// TIA Portal project "Course Work Conveyor" (V15)

(* hardware
DEVICE "S7-1200 station_1"  S7-1200 Station
   slot 0: "Rack_0"  S7-1200 Rack  Rack  V1.0
   slot 1: "PLC_1"  CPU 1214C DC/DC/DC  6ES7 214-1AG40-0XB0  V4.0
   slot 3: "AQ 1x12BIT_1"  AQ1 signal board  6ES7 232-4HA30-0XB0  V1.0
DEVICE "HMI_1"  KTP700 Basic PN
   slot 0: "HMI_1"  KTP700 Basic PN  6AV2 123-2GB03-0AX0  15.0.0.0
   slot 1: "HMI_RT_1"  KTP700 Basic PN  6AV2 123-2GB03-0AX0  15.0.0.0
   slot 5: "HMI_1.IE_CP_1"  PROFINET Interface  15.0.0.0
      slot 1: "PROFINET Interface_1"  PROFINET Interface
         slot 1: "Port_1"  Port
*)

// ===== PLC "PLC_1"  CPU 1214C DC/DC/DC =====

VAR_GLOBAL   // PLC tag table "Input/Output/Bit Tag Table"
   "EMS" AT %I0.0 : Bool;   // Emergency Stop Button NC (Input)
   "S1_Optical" AT %I0.1 : Bool;   // Optical Start Conveyor Sensor - NO (Input)
   "S2_Optical" AT %I0.2 : Bool;   // Optical Check Size Sensor NO (Input)
   "S3_Heat_or_Reject" AT %I0.3 : Bool;   // Optical Heat or Reject position Sensor NO (Input)
   "Temperature_Read_in" AT %IW64 : Int;   // Analogue Temperature (Input)
   "Reject" AT %Q0.0 : Bool;   // Rejection Solenoid (Output)
   "Conveyor" AT %Q0.1 : Bool;   // Conveyor Run (Output)
   "Furnace" AT %Q0.2 : Bool;   // Furnace Heater (Output)
   "System_Enable" AT %M0.0 : Bool;   // System Enable (Bit)
   "Detected_Large" AT %M0.1 : Bool;   // Large piece (Detected) (Bit)
   "Detected_Small" AT %M0.2 : Bool;   // Small piece (Detected) (Bit)
   "Reject_for_Large" AT %M0.5 : Bool;   // Large Rejection (Selected) (Bit)
   "Reject_for_Small" AT %M0.4 : Bool;   // Small Rejection (Selected) (Bit)
   "Furnace_Enable" AT %M0.6 : Bool;   // Furnace conditions met (Bit)
   "Piece_Size_Reset" AT %M0.7 : Bool;   // Reset the basket size (Bit)
   "PV_Memory" AT %MD1 : Real;   // Present Value reading word (Word byte)
   "Temp_in_Range" AT %M11.0 : Bool;   // Temperature in Range Confirmation (Bit)
   "Auto_Stop_Reset" AT %M11.2 : Bool;   // Automatic Stop and Reset for errors (Bit)
   "Temp_High_Alarm" AT %M11.3 : Bool;   // Furnace Alarm Temperature too High (Bit)
   "Temp_Low_Alarm" AT %M11.4 : Bool;   // Furnace Alarm Temperature too Low (Bit)
   "Temp_High_Set_Point" AT %MD12 : Real;   // High Temperature Setpoint (Bit)
   "Temp_Low_Set_Point" AT %MD16 : Real;   // Low Temperature Setpoint (Bit)
   "Temp_Limit_High_Range" AT %MD20 : Real;   // Temperature range confirmation High (Bit)
   "Temp_Limit_Low_Range" AT %MD24 : Real;   // Temperature range confirmation Low (Bit)
   "Furnace_Cycle_end" AT %M28.0 : Bool;   // End of Furnace cycle (Bit)
   "Piece_selected" AT %M28.3 : Bool;   // Confirms a piece size has been selected. (Bit)
   "Piece_Detected" AT %M28.4 : Bool;   // Confirms a piece has been detected.(Bit)
   "Counter_Reset_Large" AT %M28.5 : Bool;   // Large Piece Counter Reset (Bit)
   "Counter_Reset_Small" AT %M28.6 : Bool;   // Small Piece Counter Reset (Bit)
   "Counter_Reset_Errors" AT %M28.7 : Bool;   // Error Counter Reset (Bit)
   "Counter_Reset_Rejects" AT %M29.0 : Bool;   // Piece Reject Counter Reset (Bit)
END_VAR

VAR_GLOBAL   // PLC tag table "HMI Control Tag Table"
   "PB_Furnace_Activation_HMI" AT %M10.7 : Bool;   // Push Button: to Activate PID control of Furnace NO (Input)
   "PB_Small_HMI" AT %M10.0 : Bool;   // Push Button: Small Size reject NO (Input)
   "PB_Large_HMI" AT %M10.2 : Bool;   // Push Button: Large Size reject NO (Input)
   "PB_Manual_HMI" AT %M10.3 : Bool;   // Push Button: Mode Manual Selected NO (Input)
   "PB_Automatic_HMI" AT %M10.4 : Bool;   // Push Button: Mode Automatic Selected NO (Input)
   "PB_Reject_All_HMI" AT %M10.5 : Bool;   // Push Button: Reject All Size of Pieces NO (Input)
   "PB_Stop_Reset_HMI" AT %M10.6 : Bool;   // Push Button: Stop/Reset process cycle NO (Input)
   "PB_Furnace_Deactivation_HMI" AT %M11.1 : Bool;   // Push Button: to deactivate PID control of Furnace NO (Input)
   "PB_Reset_Counter_Large_HMI" AT %M11.5 : Bool;   // Push Button: to reset the large piece counter NO (Input)
   "PB_Reset_Counter_Small_HMI" AT %M11.6 : Bool;   // Push Button: to reset the small piece counter NO (Input)
   "PB_Reset_Counter_Errors_HMI" AT %M11.7 : Bool;   // Push Button: to reset the error counter NO (Input)
   "PB_Reset_Counter_Rejects_HMI" AT %M28.1 : Bool;   // Push Button: to reset the rejects counter NO (Input)
   "PB_Reset_Counter_All_HMI" AT %M28.2 : Bool;   // Push Button: to reset all the counters NO (Input)
   "Piece_inserted_Error_Light_HMI" AT %M29.1 : Bool;   // Error Light on HMI for Piece inserted before end the of cycle (Output)
END_VAR

DATA_BLOCK "Temp_Analog_In_DB"   // DB2
{ S7_Optimized_Access := 'TRUE' }
VERSION : 0.1
// stored: InstanceOfName Temp_Analog_In
"Temp_Analog_In"
BEGIN
END_DATA_BLOCK

// folder: System blocks/Program resources

DATA_BLOCK "Piece_Size_Reset_Delay_Timer_0_DB_2"   // DB3
{ S7_Optimized_Access := 'TRUE' }
AUTHOR : Simatic
FAMILY : IEC
NAME : IEC_TMR
VERSION : 1.0
// stored: InstanceOfName IEC_TIMER
"IEC_TIMER"
BEGIN
END_DATA_BLOCK

DATA_BLOCK "Small_Piece_Counter_0_DB"   // DB7
{ S7_Optimized_Access := 'TRUE' }
AUTHOR : Simatic
FAMILY : IEC
NAME : CNTR
VERSION : 1.0
// stored: InstanceOfName IEC_COUNTER
"IEC_COUNTER"
BEGIN
END_DATA_BLOCK

DATA_BLOCK "Large_Piece_Counter_0_DB"   // DB8
{ S7_Optimized_Access := 'TRUE' }
AUTHOR : Simatic
FAMILY : IEC
NAME : CNTR
VERSION : 1.0
// stored: InstanceOfName IEC_COUNTER
"IEC_COUNTER"
BEGIN
END_DATA_BLOCK

DATA_BLOCK "Furnace_Timer_0_DB_2"   // DB9
{ S7_Optimized_Access := 'TRUE' }
AUTHOR : Simatic
FAMILY : IEC
NAME : IEC_TMR
VERSION : 1.0
// stored: InstanceOfName IEC_TIMER
"IEC_TIMER"
BEGIN
END_DATA_BLOCK

DATA_BLOCK "Total_Error_Counter_0_DB"   // DB10
{ S7_Optimized_Access := 'TRUE' }
AUTHOR : Simatic
FAMILY : IEC
NAME : CNTR
VERSION : 1.0
// stored: InstanceOfName IEC_COUNTER
"IEC_COUNTER"
BEGIN
END_DATA_BLOCK

DATA_BLOCK "Total_Piece_Reject_Counter_0_DB"   // DB11
{ S7_Optimized_Access := 'TRUE' }
AUTHOR : Simatic
FAMILY : IEC
NAME : CNTR
VERSION : 1.0
// stored: InstanceOfName IEC_COUNTER
"IEC_COUNTER"
BEGIN
END_DATA_BLOCK

DATA_BLOCK "Reject_on_Error_Delay_Timer_0_DB_3"   // DB12
{ S7_Optimized_Access := 'TRUE' }
AUTHOR : Simatic
FAMILY : IEC
NAME : IEC_TMR
VERSION : 1.0
// stored: InstanceOfName IEC_TIMER
"IEC_TIMER"
BEGIN
END_DATA_BLOCK

// folder: (top level)

FUNCTION_BLOCK "Temp_Analog_In"   // FB1, LAD
{ S7_Optimized_Access := 'TRUE' }
VERSION : 0.1
// Function Block: Temperature (Analogue Signal In). 
// The Temperature signal is read, normalised and then put to scale.
   VAR_INPUT
      ChannelAddress : Int;
      HR : Real;
      LR : Real;
   END_VAR
   VAR_IN_OUT
      PV : Real;   // Input reading
   END_VAR
   VAR_TEMP
      Normalised : Real;   // Normalise Temperature Value
   END_VAR
BEGIN

REGION Network 1: Value Normalising.
   // Normalising reading values (Scale 0 to 27648).
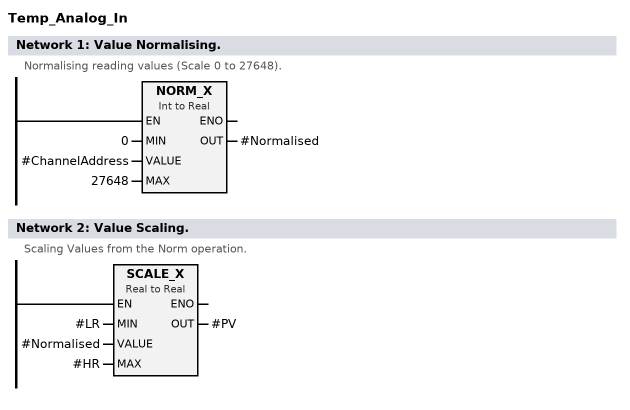
   RUNG wire#powerrail
      { S7_Templates := "[SrcType := Int, DestType := Real]" } Normalize(min := 0, value := #ChannelAddress, max := 27648, out => #Normalised)
   END_RUNG
   // the same network as SCL:
   #Normalised := NORM_X(MIN := 0, VALUE := #ChannelAddress, MAX := 27648);
END_REGION

REGION Network 2: Value Scaling.
   // Scaling Values from the Norm operation.
   RUNG wire#powerrail
      { S7_Templates := "[SrcType := Real, DestType := Real]" } Scale(min := #LR, value := #Normalised, max := #HR, out => #PV)
   END_RUNG
   // the same network as SCL:
   #PV := SCALE_X(MIN := #LR, VALUE := #Normalised, MAX := #HR);
END_REGION
END_FUNCTION_BLOCK

FUNCTION "Conveyor Belt" : Void   // FC1, LAD
{ S7_Optimized_Access := 'TRUE' }
VERSION : 0.1
// Conveyor Related Operations:
// Conveyor Run.
// Piece Size Detection.
// Piece size Confirmation.
// Rejection Solenoid.
// Enable Furnace Operation.
// Furnace in Operation.
// Basket Size Reset.
BEGIN

REGION Network 1: Conveyor Run
   // Once size is selected AND System is Enabled (Automatic mode) OR Manual == Conveyor ON
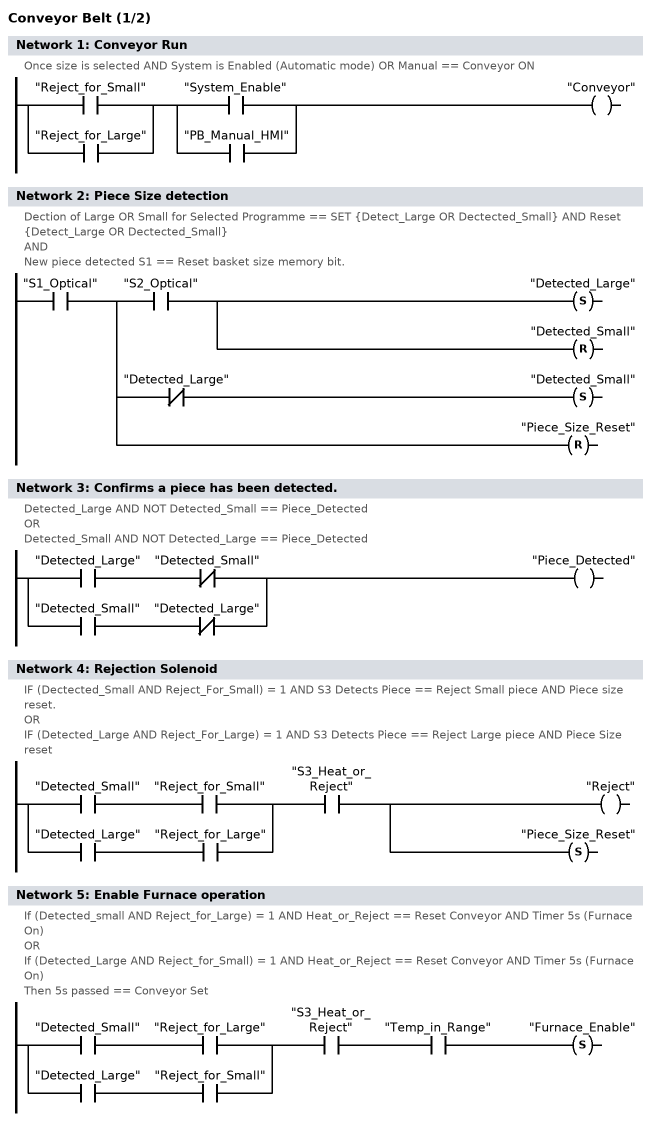
   RUNG wire#powerrail
      Contact( "Reject_for_Small" )
      wire#w1
      Contact( "System_Enable" )
      wire#w2
      Coil( "Conveyor" )
   END_RUNG
   RUNG wire#powerrail
      Contact( "Reject_for_Large" )
   END_RUNG wire#w1
   RUNG wire#w1
      Contact( "PB_Manual_HMI" )
   END_RUNG wire#w2
   // the same network as SCL:
   "Conveyor" := ("Reject_for_Small" OR "Reject_for_Large") AND ("System_Enable" OR "PB_Manual_HMI");
END_REGION

REGION Network 2: Piece Size detection
   // Dection of Large OR Small for Selected Programme == SET {Detect_Large OR Dectected_Small} AND Reset {Detect_Large OR Dectected_Small}
   // AND
   // New piece detected S1 == Reset basket size memory bit.
   RUNG wire#powerrail
      Contact( "S1_Optical" )
      wire#w1
      Contact( "S2_Optical" )
      wire#w2
      S_Coil( "Detected_Large" )
   END_RUNG
   RUNG wire#w2
      R_Coil( "Detected_Small" )
   END_RUNG
   RUNG wire#w1
      I_Contact( "Detected_Large" )
      S_Coil( "Detected_Small" )
   END_RUNG
   RUNG wire#w1
      R_Coil( "Piece_Size_Reset" )
   END_RUNG
   // the same network as SCL:
   IF "S1_Optical" AND "S2_Optical" THEN
       "Detected_Large" := TRUE;
       "Detected_Small" := FALSE;
   END_IF;
   IF "S1_Optical" AND NOT "Detected_Large" THEN "Detected_Small" := TRUE; END_IF;
   IF "S1_Optical" THEN "Piece_Size_Reset" := FALSE; END_IF;
END_REGION

REGION Network 3: Confirms a piece has been detected.
   // Detected_Large AND NOT Detected_Small == Piece_Detected
   // OR
   // Detected_Small AND NOT Detected_Large == Piece_Detected
   RUNG wire#powerrail
      Contact( "Detected_Large" )
      I_Contact( "Detected_Small" )
      wire#w1
      Coil( "Piece_Detected" )
   END_RUNG
   RUNG wire#powerrail
      Contact( "Detected_Small" )
      I_Contact( "Detected_Large" )
   END_RUNG wire#w1
   // the same network as SCL:
   "Piece_Detected" := ("Detected_Large" AND NOT "Detected_Small") OR ("Detected_Small" AND NOT "Detected_Large");
END_REGION

REGION Network 4: Rejection Solenoid
   // IF (Dectected_Small AND Reject_For_Small) = 1 AND S3 Detects Piece == Reject Small piece AND Piece size reset.
   // OR
   // IF (Detected_Large AND Reject_For_Large) = 1 AND S3 Detects Piece == Reject Large piece AND Piece Size reset
   RUNG wire#powerrail
      Contact( "Detected_Small" )
      Contact( "Reject_for_Small" )
      wire#w1
      Contact( "S3_Heat_or_Reject" )
      wire#w2
      Coil( "Reject" )
   END_RUNG
   RUNG wire#powerrail
      Contact( "Detected_Large" )
      Contact( "Reject_for_Large" )
   END_RUNG wire#w1
   RUNG wire#w2
      S_Coil( "Piece_Size_Reset" )
   END_RUNG
   // the same network as SCL:
   "Reject" := (("Detected_Small" AND "Reject_for_Small") OR ("Detected_Large" AND "Reject_for_Large")) AND "S3_Heat_or_Reject";
   IF "Reject" THEN "Piece_Size_Reset" := TRUE; END_IF;
END_REGION

REGION Network 5: Enable Furnace operation
   // If (Detected_small AND Reject_for_Large) = 1 AND Heat_or_Reject == Reset Conveyor AND Timer 5s (Furnace On)
   // OR
   // If (Detected_Large AND Reject_for_Small) = 1 AND Heat_or_Reject == Reset Conveyor AND Timer 5s (Furnace On)
   // Then 5s passed == Conveyor Set
   RUNG wire#powerrail
      Contact( "Detected_Small" )
      Contact( "Reject_for_Large" )
      wire#w1
      Contact( "S3_Heat_or_Reject" )
      Contact( "Temp_in_Range" )
      S_Coil( "Furnace_Enable" )
   END_RUNG
   RUNG wire#powerrail
      Contact( "Detected_Large" )
      Contact( "Reject_for_Small" )
   END_RUNG wire#w1
   // the same network as SCL:
   IF (("Detected_Small" AND "Reject_for_Large") OR ("Detected_Large" AND "Reject_for_Small")) AND "S3_Heat_or_Reject" AND "Temp_in_Range" THEN
       "Furnace_Enable" := TRUE;
   END_IF;
END_REGION

REGION Network 6: Furnace in Operation
   // IF Furnace enabled == stop Conveyor 
   // THEN  Temp_in_Range == start 5s Timer
   // AND THEN at 5s == reset Conveyor AND Reset_Piece_Size AND SET  Furnace_Cycle_end
   // Note: Timer delay on piece size reset to allow and of cycle tasks before new cycle.
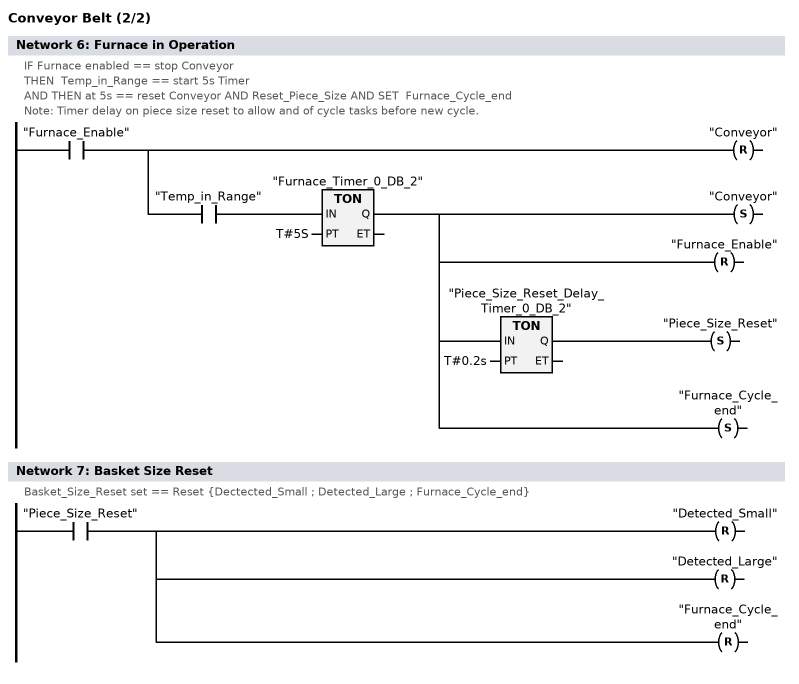
   IF "Furnace_Enable" THEN "Conveyor" := FALSE; END_IF;
   "Furnace_Timer_0_DB_2".TON(IN := "Furnace_Enable" AND "Temp_in_Range", PT := T#5S);
   IF "Furnace_Timer_0_DB_2".Q THEN
       "Conveyor" := TRUE;
       "Furnace_Enable" := FALSE;
   END_IF;
   "Piece_Size_Reset_Delay_Timer_0_DB_2".TON(IN := "Furnace_Timer_0_DB_2".Q, PT := T#0.2s);
   IF "Piece_Size_Reset_Delay_Timer_0_DB_2".Q THEN "Piece_Size_Reset" := TRUE; END_IF;
   IF "Furnace_Timer_0_DB_2".Q THEN "Furnace_Cycle_end" := TRUE; END_IF;
END_REGION

REGION Network 7: Basket Size Reset
   // Basket_Size_Reset set == Reset {Dectected_Small ; Detected_Large ; Furnace_Cycle_end}
   RUNG wire#powerrail
      Contact( "Piece_Size_Reset" )
      wire#w1
      R_Coil( "Detected_Small" )
   END_RUNG
   RUNG wire#w1
      R_Coil( "Detected_Large" )
   END_RUNG
   RUNG wire#w1
      R_Coil( "Furnace_Cycle_end" )
   END_RUNG
   // the same network as SCL:
   IF "Piece_Size_Reset" THEN
       "Detected_Small" := FALSE;
       "Detected_Large" := FALSE;
       "Furnace_Cycle_end" := FALSE;
   END_IF;
END_REGION
END_FUNCTION

FUNCTION "Temperature Function" : Void   // FC2, LAD
{ S7_Optimized_Access := 'TRUE' }
VERSION : 0.1
BEGIN

REGION Network 1: PID Control of the Furnace Activation/Deactivation
   // IF Button "Funace Activation" pressed == PID Control ON
   // OR
   // IF Button "Stop Furnace" pressed == PID Control OFF
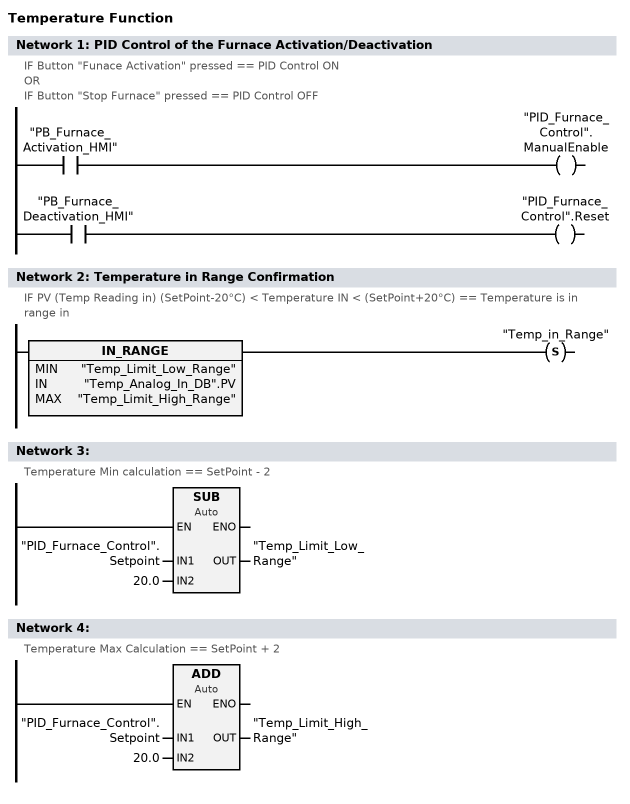
   RUNG wire#powerrail
      Contact( "PB_Furnace_Activation_HMI" )
      Coil( "PID_Furnace_Control".ManualEnable )
   END_RUNG
   RUNG wire#powerrail
      Contact( "PB_Furnace_Deactivation_HMI" )
      Coil( "PID_Furnace_Control".Reset )
   END_RUNG
   // the same network as SCL:
   "PID_Furnace_Control".ManualEnable := "PB_Furnace_Activation_HMI";
   "PID_Furnace_Control".Reset := "PB_Furnace_Deactivation_HMI";
END_REGION

REGION Network 2: Temperature in Range Confirmation
   // IF PV (Temp Reading in) (SetPoint-20°C) < Temperature IN < (SetPoint+20°C) == Temperature is in range in
   RUNG wire#powerrail
      { S7_Templates := "SrcType := Real" } InRange(min := "Temp_Limit_Low_Range", in := "Temp_Analog_In_DB".PV, max := "Temp_Limit_High_Range")
      S_Coil( "Temp_in_Range" )
   END_RUNG
   // the same network as SCL:
   IF ("Temp_Limit_Low_Range" <= "Temp_Analog_In_DB".PV) AND ("Temp_Analog_In_DB".PV <= "Temp_Limit_High_Range") THEN
       "Temp_in_Range" := TRUE;
   END_IF;
END_REGION

REGION Network 3
   // Temperature Min calculation == SetPoint - 2
   RUNG wire#powerrail
      Sub(in1 := "PID_Furnace_Control".Setpoint, in2 := 20.0, out => "Temp_Limit_Low_Range")
   END_RUNG
   // the same network as SCL:
   "Temp_Limit_Low_Range" := "PID_Furnace_Control".Setpoint - 20.0;
END_REGION

REGION Network 4
   // Temperature Max Calculation == SetPoint + 2
   RUNG wire#powerrail
      Add(in1 := "PID_Furnace_Control".Setpoint, in2 := 20.0, out => "Temp_Limit_High_Range")
   END_RUNG
   // the same network as SCL:
   "Temp_Limit_High_Range" := "PID_Furnace_Control".Setpoint + 20.0;
END_REGION
END_FUNCTION

FUNCTION "Error_Handling" : Void   // FC3, LAD
{ S7_Optimized_Access := 'TRUE' }
VERSION : 0.1
// Error Handling Function:
// Piece inserted before end of previous cycle
// Temperature is Too HIGH or too LOW.
   VAR_TEMP   // added for the SCL form of the ladder/FBD networks
      _w1 : Bool;
   END_VAR
BEGIN

REGION Network 1: Rejection Solenoid
   // Piece inserted before end of previous cycle:
   // Piece detected at Heating/Rejection point AND (S1 OR S2) triggered == Reject Part AND Stop/Reset Cycle AND Sets the Error Light ON on the HMI.
   // Note: The Timer delays the reject to leave time for Auto_Stop_Reset and the Error Light to set ON.
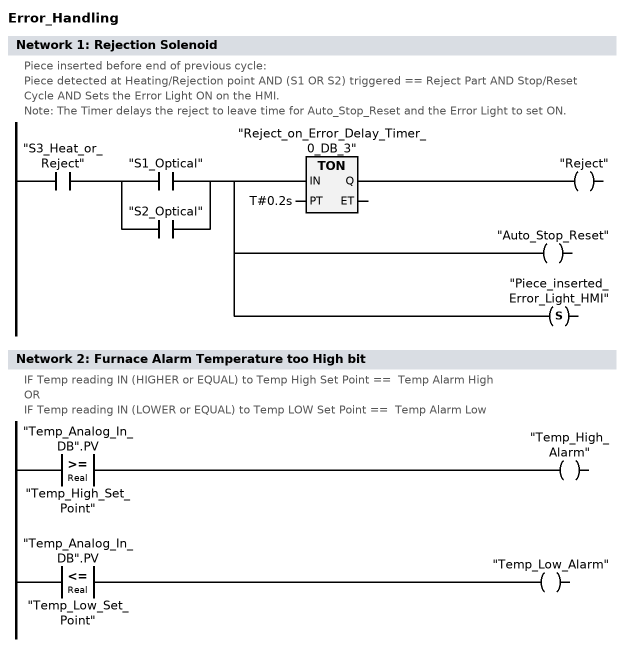
   #_w1 := "S3_Heat_or_Reject" AND ("S1_Optical" OR "S2_Optical");
   "Reject_on_Error_Delay_Timer_0_DB_3".TON(IN := #_w1, PT := T#0.2s);
   "Reject" := "Reject_on_Error_Delay_Timer_0_DB_3".Q;
   "Auto_Stop_Reset" := #_w1;
   IF #_w1 THEN "Piece_inserted_Error_Light_HMI" := TRUE; END_IF;
END_REGION

REGION Network 2: Furnace Alarm Temperature too High bit
   // IF Temp reading IN (HIGHER or EQUAL) to Temp High Set Point ==  Temp Alarm High
   // OR
   // IF Temp reading IN (LOWER or EQUAL) to Temp LOW Set Point ==  Temp Alarm Low
   RUNG wire#powerrail
      { S7_Templates := "SrcType := Real" } GE_Contact(in1 := "Temp_Analog_In_DB".PV, in2 := "Temp_High_Set_Point")
      Coil( "Temp_High_Alarm" )
   END_RUNG
   RUNG wire#powerrail
      { S7_Templates := "SrcType := Real" } LE_Contact(in1 := "Temp_Analog_In_DB".PV, in2 := "Temp_Low_Set_Point")
      Coil( "Temp_Low_Alarm" )
   END_RUNG
   // the same network as SCL:
   "Temp_High_Alarm" := "Temp_Analog_In_DB".PV >= "Temp_High_Set_Point";
   "Temp_Low_Alarm" := "Temp_Analog_In_DB".PV <= "Temp_Low_Set_Point";
END_REGION
END_FUNCTION

FUNCTION "Counters" : Void   // FC4, LAD
{ S7_Optimized_Access := 'TRUE' }
VERSION : 0.1
// Counters in the process for each manufactured parts and for the number of errors.
BEGIN

REGION Network 1: Large part manufactured counter.
   // IF Detected_Large AND Reject_for_small AND Furnace_Cycle_end == Counter +1
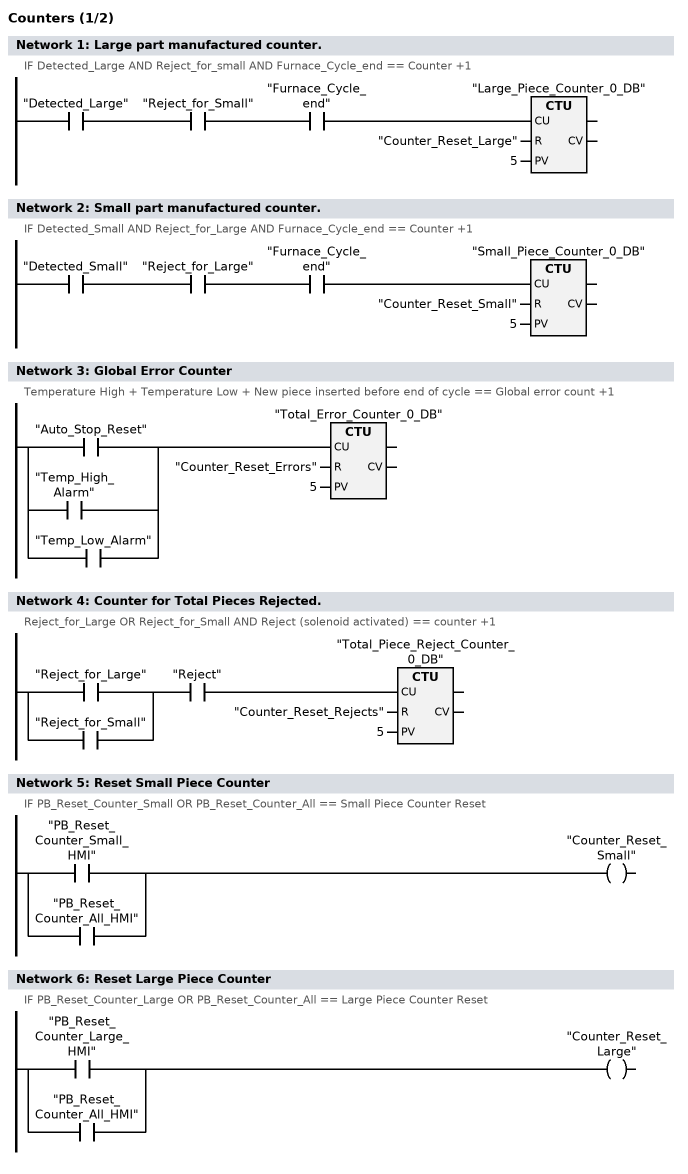
   "Large_Piece_Counter_0_DB".CTU(CU := "Detected_Large" AND "Reject_for_Small" AND "Furnace_Cycle_end",
                           R := "Counter_Reset_Large",
                           PV := 5);
END_REGION

REGION Network 2: Small part manufactured counter.
   // IF Detected_Small AND Reject_for_Large AND Furnace_Cycle_end == Counter +1
   "Small_Piece_Counter_0_DB".CTU(CU := "Detected_Small" AND "Reject_for_Large" AND "Furnace_Cycle_end",
                           R := "Counter_Reset_Small",
                           PV := 5);
END_REGION

REGION Network 3: Global Error Counter
   // Temperature High + Temperature Low + New piece inserted before end of cycle == Global error count +1
   "Total_Error_Counter_0_DB".CTU(CU := "Auto_Stop_Reset" OR "Temp_High_Alarm" OR "Temp_Low_Alarm",
                           R := "Counter_Reset_Errors",
                           PV := 5);
END_REGION

REGION Network 4: Counter for Total Pieces Rejected.
   // Reject_for_Large OR Reject_for_Small AND Reject (solenoid activated) == counter +1
   "Total_Piece_Reject_Counter_0_DB".CTU(CU := ("Reject_for_Large" OR "Reject_for_Small") AND "Reject",
                           R := "Counter_Reset_Rejects",
                           PV := 5);
END_REGION

REGION Network 5: Reset Small Piece Counter
   // IF PB_Reset_Counter_Small OR PB_Reset_Counter_All == Small Piece Counter Reset
   RUNG wire#powerrail
      Contact( "PB_Reset_Counter_Small_HMI" )
      wire#w1
      Coil( "Counter_Reset_Small" )
   END_RUNG
   RUNG wire#powerrail
      Contact( "PB_Reset_Counter_All_HMI" )
   END_RUNG wire#w1
   // the same network as SCL:
   "Counter_Reset_Small" := "PB_Reset_Counter_Small_HMI" OR "PB_Reset_Counter_All_HMI";
END_REGION

REGION Network 6: Reset Large Piece Counter
   // IF PB_Reset_Counter_Large OR PB_Reset_Counter_All == Large Piece Counter Reset
   RUNG wire#powerrail
      Contact( "PB_Reset_Counter_Large_HMI" )
      wire#w1
      Coil( "Counter_Reset_Large" )
   END_RUNG
   RUNG wire#powerrail
      Contact( "PB_Reset_Counter_All_HMI" )
   END_RUNG wire#w1
   // the same network as SCL:
   "Counter_Reset_Large" := "PB_Reset_Counter_Large_HMI" OR "PB_Reset_Counter_All_HMI";
END_REGION

REGION Network 7: Reset Rejected Piece Counter
   // IF PB_Reset_Counter_Reject OR PB_Reset_Counter_All == Total Piece Rejects Counter Reset
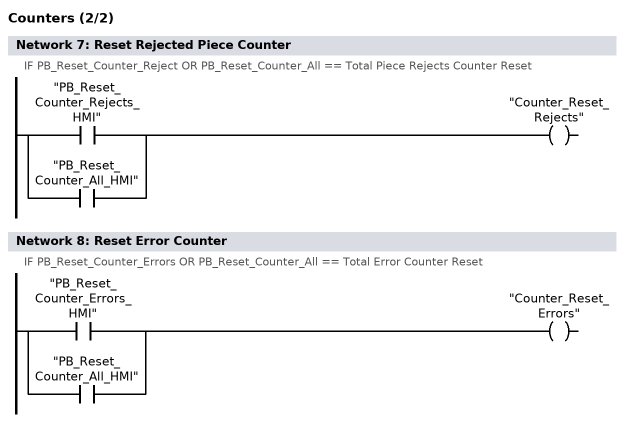
   RUNG wire#powerrail
      Contact( "PB_Reset_Counter_Rejects_HMI" )
      wire#w1
      Coil( "Counter_Reset_Rejects" )
   END_RUNG
   RUNG wire#powerrail
      Contact( "PB_Reset_Counter_All_HMI" )
   END_RUNG wire#w1
   // the same network as SCL:
   "Counter_Reset_Rejects" := "PB_Reset_Counter_Rejects_HMI" OR "PB_Reset_Counter_All_HMI";
END_REGION

REGION Network 8: Reset Error Counter
   // IF PB_Reset_Counter_Errors OR PB_Reset_Counter_All == Total Error Counter Reset
   RUNG wire#powerrail
      Contact( "PB_Reset_Counter_Errors_HMI" )
      wire#w1
      Coil( "Counter_Reset_Errors" )
   END_RUNG
   RUNG wire#powerrail
      Contact( "PB_Reset_Counter_All_HMI" )
   END_RUNG wire#w1
   // the same network as SCL:
   "Counter_Reset_Errors" := "PB_Reset_Counter_Errors_HMI" OR "PB_Reset_Counter_All_HMI";
END_REGION
END_FUNCTION

FUNCTION "System_Controls" : Void   // FC5, LAD
TITLE = Systems_Controls
{ S7_Optimized_Access := 'TRUE' }
VERSION : 0.1
// Interface controls to enable the automatic mode.
// Stop/Reset on HMI and auto Reset operations.
// Piece size selection and confirmation operation.
BEGIN

REGION Network 1: Automatic Mode System Enable
   // Automatic Mode && Part Detected AND Temp in Range AND NOT Manual mode  == System enabled AND Error_Light for piece inserted reset.
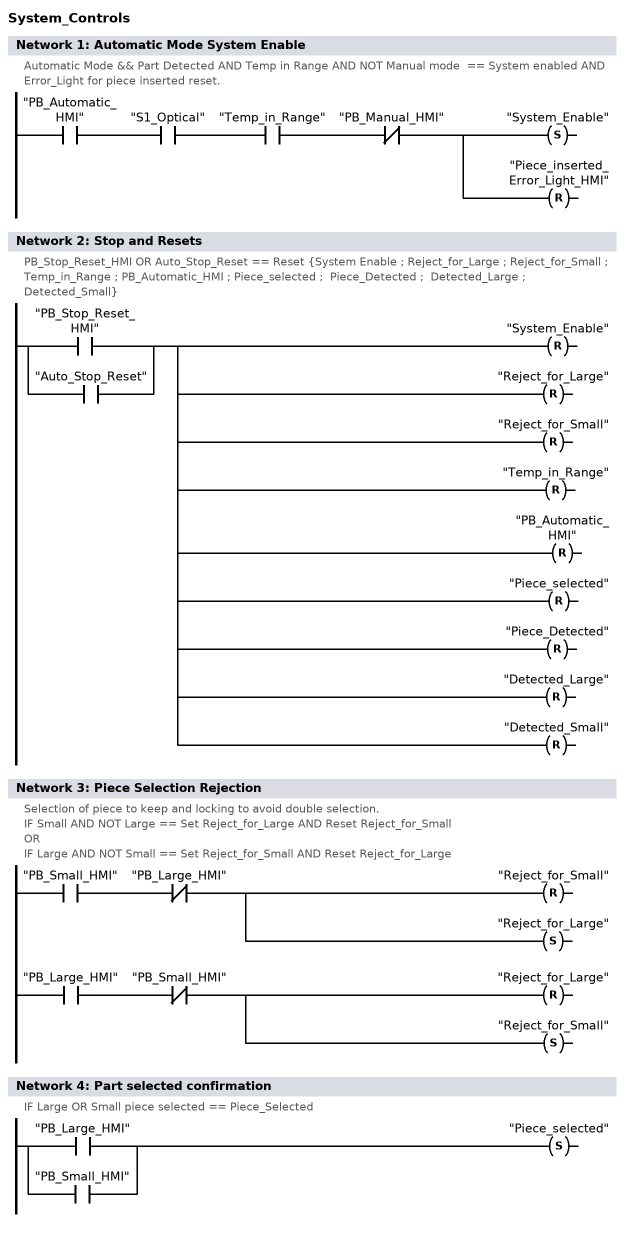
   RUNG wire#powerrail
      Contact( "PB_Automatic_HMI" )
      Contact( "S1_Optical" )
      Contact( "Temp_in_Range" )
      I_Contact( "PB_Manual_HMI" )
      wire#w1
      S_Coil( "System_Enable" )
   END_RUNG
   RUNG wire#w1
      R_Coil( "Piece_inserted_Error_Light_HMI" )
   END_RUNG
   // the same network as SCL:
   IF "PB_Automatic_HMI" AND "S1_Optical" AND "Temp_in_Range" AND NOT "PB_Manual_HMI" THEN
       "System_Enable" := TRUE;
       "Piece_inserted_Error_Light_HMI" := FALSE;
   END_IF;
END_REGION

REGION Network 2: Stop and Resets
   // PB_Stop_Reset_HMI OR Auto_Stop_Reset == Reset {System Enable ; Reject_for_Large ; Reject_for_Small ; Temp_in_Range ; PB_Automatic_HMI ; Piece_selected ;  Piece_Detected ;  Detected_Large ; Detected_Small}
   RUNG wire#powerrail
      Contact( "PB_Stop_Reset_HMI" )
      wire#w1
      R_Coil( "System_Enable" )
   END_RUNG
   RUNG wire#powerrail
      Contact( "Auto_Stop_Reset" )
   END_RUNG wire#w1
   RUNG wire#w1
      R_Coil( "Reject_for_Large" )
   END_RUNG
   RUNG wire#w1
      R_Coil( "Reject_for_Small" )
   END_RUNG
   RUNG wire#w1
      R_Coil( "Temp_in_Range" )
   END_RUNG
   RUNG wire#w1
      R_Coil( "PB_Automatic_HMI" )
   END_RUNG
   RUNG wire#w1
      R_Coil( "Piece_selected" )
   END_RUNG
   RUNG wire#w1
      R_Coil( "Piece_Detected" )
   END_RUNG
   RUNG wire#w1
      R_Coil( "Detected_Large" )
   END_RUNG
   RUNG wire#w1
      R_Coil( "Detected_Small" )
   END_RUNG
   // the same network as SCL:
   IF "PB_Stop_Reset_HMI" OR "Auto_Stop_Reset" THEN
       "System_Enable" := FALSE;
       "Reject_for_Large" := FALSE;
       "Reject_for_Small" := FALSE;
       "Temp_in_Range" := FALSE;
       "PB_Automatic_HMI" := FALSE;
       "Piece_selected" := FALSE;
       "Piece_Detected" := FALSE;
       "Detected_Large" := FALSE;
       "Detected_Small" := FALSE;
   END_IF;
END_REGION

REGION Network 3: Piece Selection Rejection
   // Selection of piece to keep and locking to avoid double selection. 
   // IF Small AND NOT Large == Set Reject_for_Large AND Reset Reject_for_Small
   // OR
   // IF Large AND NOT Small == Set Reject_for_Small AND Reset Reject_for_Large
   RUNG wire#powerrail
      Contact( "PB_Small_HMI" )
      I_Contact( "PB_Large_HMI" )
      wire#w1
      R_Coil( "Reject_for_Small" )
   END_RUNG
   RUNG wire#w1
      S_Coil( "Reject_for_Large" )
   END_RUNG
   RUNG wire#powerrail
      Contact( "PB_Large_HMI" )
      I_Contact( "PB_Small_HMI" )
      wire#w2
      R_Coil( "Reject_for_Large" )
   END_RUNG
   RUNG wire#w2
      S_Coil( "Reject_for_Small" )
   END_RUNG
   // the same network as SCL:
   IF "PB_Small_HMI" AND NOT "PB_Large_HMI" THEN
       "Reject_for_Small" := FALSE;
       "Reject_for_Large" := TRUE;
   END_IF;
   IF "PB_Large_HMI" AND NOT "PB_Small_HMI" THEN
       "Reject_for_Large" := FALSE;
       "Reject_for_Small" := TRUE;
   END_IF;
END_REGION

REGION Network 4: Part selected confirmation
   // IF Large OR Small piece selected == Piece_Selected
   RUNG wire#powerrail
      Contact( "PB_Large_HMI" )
      wire#w1
      S_Coil( "Piece_selected" )
   END_RUNG
   RUNG wire#powerrail
      Contact( "PB_Small_HMI" )
   END_RUNG wire#w1
   // the same network as SCL:
   IF "PB_Large_HMI" OR "PB_Small_HMI" THEN "Piece_selected" := TRUE; END_IF;
END_REGION
END_FUNCTION

ORGANIZATION_BLOCK "Main"   // OB1, LAD, ProgramCycle
TITLE = "Main Program Sweep (Cycle)"
{ S7_Optimized_Access := 'TRUE' }
VERSION : 0.1
// Main loop of the Programme. It contains:
// The System Controls and Conveyor Belt operation
// The read in value from the analogue temperature sensor.
// The Counter function.
   VAR_INPUT
      Initial_Call : Bool;   // Initial call of this OB
      Remanence : Bool;   // =True, if remanent data are available
   END_VAR
   VAR_TEMP   // added for the SCL form of the ladder/FBD networks
      _w1 : Bool;
   END_VAR
BEGIN

REGION Network 1: Programme main functions
   // System_Controls: Link with the HMI interface.  Allows piece sizes selection and programme selection (Automatic or Manual)
   // Conveyor Belt:  Conveyor belt, piece rejection and furnace operation.
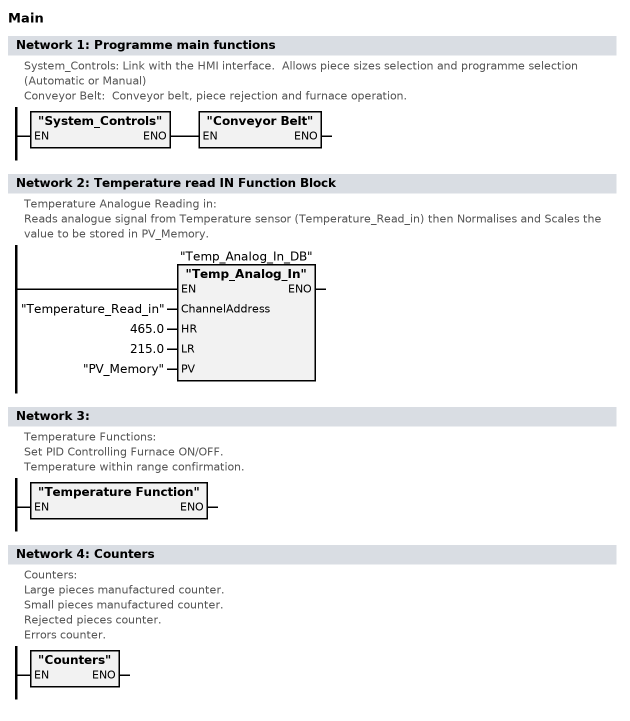
   RUNG wire#powerrail
      "System_Controls"()
      "Conveyor Belt"()
   END_RUNG
   // the same network as SCL:
   "System_Controls"(ENO => #_w1);
   IF #_w1 THEN "Conveyor Belt"(); END_IF;
END_REGION

REGION Network 2: Temperature read IN Function Block
   // Temperature Analogue Reading in:
   // Reads analogue signal from Temperature sensor (Temperature_Read_in) then Normalises and Scales the value to be stored in PV_Memory.
   RUNG wire#powerrail
      "Temp_Analog_In_DB"(ChannelAddress := "Temperature_Read_in", HR := 465.0, LR := 215.0, PV := "PV_Memory")
   END_RUNG
   // the same network as SCL:
   "Temp_Analog_In_DB"(ChannelAddress := "Temperature_Read_in", HR := 465.0, LR := 215.0, PV := "PV_Memory");   // "Temp_Analog_In"
END_REGION

REGION Network 3
   // Temperature Functions: 
   // Set PID Controlling Furnace ON/OFF.
   // Temperature within range confirmation.
   RUNG wire#powerrail
      "Temperature Function"()
   END_RUNG
   // the same network as SCL:
   "Temperature Function"();
END_REGION

REGION Network 4: Counters
   // Counters:
   // Large pieces manufactured counter.
   // Small pieces manufactured counter.
   // Rejected pieces counter.
   // Errors counter.
   RUNG wire#powerrail
      "Counters"()
   END_RUNG
   // the same network as SCL:
   "Counters"();
END_REGION
END_ORGANIZATION_BLOCK

ORGANIZATION_BLOCK "Cyclic interrupt"   // OB30, LAD, CyclicInterrupt
{ S7_Optimized_Access := 'TRUE' }
VERSION : 0.1
// OB30 allows for background tasks to run at the same time time as the main programme:
// Furnace PID Control.
// Error Handling function.
   VAR_INPUT
      Initial_Call : Bool;   // Initial call of this OB
      Event_Count : Int;   // Events discarded
   END_VAR
BEGIN

REGION Network 1: PID Furnace Control
   // PID is set ON by PB_Funace_Activation_HMI on ManualEnable.
   // PID is set OFF by PB_Furnace_Deactivation_HMI on Reset.
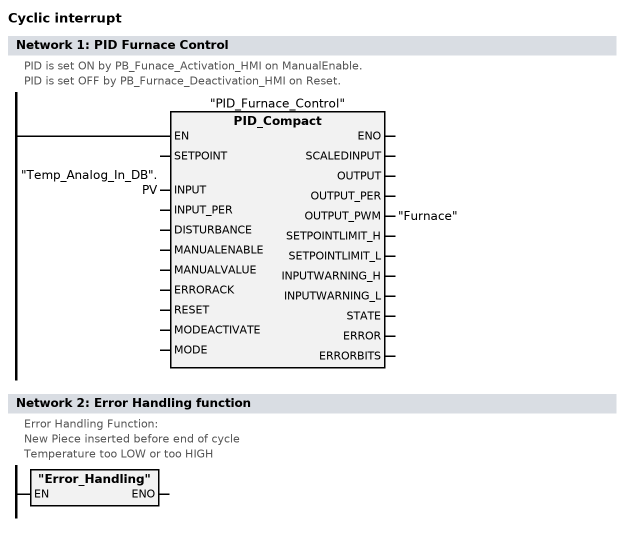
   "PID_Furnace_Control"(Input := "Temp_Analog_In_DB".PV, Output_PWM => "Furnace");   // PID_Compact
END_REGION

REGION Network 2: Error Handling function
   // Error Handling Function:
   // New Piece inserted before end of cycle
   // Temperature too LOW or too HIGH
   RUNG wire#powerrail
      "Error_Handling"()
   END_RUNG
   // the same network as SCL:
   "Error_Handling"();
END_REGION
END_ORGANIZATION_BLOCK

(* ===== HMI "HMI_RT_1" =====
system functions are stored by id; their names below are inferred from use
connection "HMI_Connection_1": ETHERNET, SMART_S7_1200_OMS

HMI tags "HMI tag table"
   "Tag_ScreenNumber" : UInt, internal
   "PB_Large_HMI" : Bool = PLC PB_Large_HMI AT %M10.2, 1 s   // Push Button: Large Size reject NO (Input)
   "PB_Small_HMI" : Bool = PLC PB_Small_HMI AT %M10.0, 1 s   // Push Button: Small Size reject NO (Input)
   "PB_Automatic_HMI" : Bool = PLC PB_Automatic_HMI AT %M10.4, 1 s   // Push Button: Mode Automatic Selected NO (Input)
   "PB_Stop_HMI" : Bool = PLC PB_Stop_Reset_HMI AT %M10.6, 1 s   // Push Button: Stop/Reset process cycle NO (Input)
   "PB_Manual_HMI" : Bool = PLC PB_Manual_HMI AT %M10.3, 1 s   // Push Button: Mode Manual Selected NO (Input)
   "PID_Furnace_Control_Setpoint" : Real = PLC PID_Furnace_Control.Setpoint, 1 s   // controller setpoint input
   "PID_Furnace_Control_ManualEnable" : Bool = PLC PID_Furnace_Control.ManualEnable, 1 s   // activate manual input to overwrite output
   "PB_Furnace_Activation" : Bool = PLC PB_Furnace_Activation_HMI AT %M10.7, 1 s   // Push Button: to Activate PID control of Furnace NO (Input)
   "PB_Furnace_Deactivation" : Bool = PLC PB_Furnace_Deactivation_HMI AT %M11.1, 1 s   // Push Button: to deactivate PID control of Furnace NO (Input)
   "PV_Memory" : Real = PLC PV_Memory AT %MD1, 1 s   // Present Value reading word (Word byte)
   "Temp_High_Set_Point" : Real = PLC Temp_High_Set_Point AT %MD12, 1 s   // High Temperature Setpoint (Bit)
   "Temp_Low_Set_Point" : Real = PLC Temp_Low_Set_Point AT %MD16, 1 s   // Low Temperature Setpoint (Bit)
   "LargePart_Counter_0_DB_CV" : Int = PLC Large_Piece_Counter_0_DB.CV, 1 s
   "SmallPart_Counter_0_DB_CV" : Int = PLC Small_Piece_Counter_0_DB.CV, 1 s
   "IEC_Total_Piece_Reject_Counter_0_DB_CV" : Int = PLC Total_Piece_Reject_Counter_0_DB.CV, 1 s
   "IEC_Total_Error_Counter_0_DB_CV" : Int = PLC Total_Error_Counter_0_DB.CV, 1 s   // Total Error counter Block (+1 for each error)
   "PB_Reset_Counter_Large" : Bool = PLC PB_Reset_Counter_Large_HMI AT %M11.5, 1 s
   "PB_Reset_Counter_Small" : Bool = PLC PB_Reset_Counter_Small_HMI AT %M11.6, 1 s   // Push Button: to reset the small piece counter NO (Input)
   "PB_Reset_Counter_Rejects" : Bool = PLC PB_Reset_Counter_Rejects_HMI AT %M28.1, 1 s   // Push Button: to reset the rejects counter NO (Input)
   "PB_Reset_Counter_Errors" : Bool = PLC PB_Reset_Counter_Errors_HMI AT %M11.7, 1 s   // Push Button: to reset the error counter NO (Input)
   "PB_Reset_Counter_All" : Bool = PLC PB_Reset_Counter_All_HMI AT %M28.2, 1 s   // Push Button: to reset all the counters NO (Input)
   "System Enable" : Bool = PLC System_Enable AT %M0.0, 1 s   // System Enable (Bit)
   "Temp_High_Alarm" : Bool = PLC Temp_High_Alarm AT %M11.3, 1 s   // Furnace Alarm Temperature too High (Bit)
   "Temp_Low_Alarm" : Bool = PLC Temp_Low_Alarm AT %M11.4, 1 s   // Furnace Alarm Temperature too Low (Bit)
   "Temp_in_Range" : Bool = PLC Temp_in_Range AT %M11.0, 1 s   // Temperature in Range Confirmation (Bit)
   "Furnace_Enable" : Bool = PLC Furnace_Enable AT %M0.6, 1 s   // Furnace conditions met (Bit)
   "Piece_selected" : Bool = PLC Piece_selected AT %M28.3, 1 s   // Confirms a piece size has been selected. (Bit)
   "Furnace_Timer_0_DB_2_IN" : Bool = PLC Furnace_Timer_0_DB_2.IN, 1 s   // Furnace timer (TON) block at 5s (timer)
   "Furnace_Cycle_end" : Bool = PLC Furnace_Cycle_end AT %M28.0, 1 s   // End of Furnace cycle (Bit)
   "Piece_Detected" : Bool = PLC Piece_Detected AT %M28.4, 1 s   // Confirms a piece has been detected.(Bit)
   "Reject" : Bool = PLC Reject AT %Q0.0, 1 s   // Rejection Solenoid (Output)
   "Temp_Analog_In_DB_PV" : Real = PLC Temp_Analog_In_DB.PV, 1 s   // Input reading Block from temperature probe (Input)
   "S1 Optical" : Bool = PLC S1_Optical AT %I0.1, 1 s   // Optical Start Conveyor Sensor - NO (Input)
   "S2 Optical" : Bool = PLC S2_Optical AT %I0.2, 1 s   // Optical Check Size Sensor NO (Input)
   "S3 Heat or Reject" : Bool = PLC S3_Heat_or_Reject AT %I0.3, 1 s   // Optical Heat or Reject position Sensor NO (Input)
   "Piece_inserted_Error_Light_HMI" : Bool = PLC Piece_inserted_Error_Light_HMI AT %M29.1, 1 s

Template "Template_1" 800x480
   Button "Exit" at 714,429 size 71x50; TextOff 'Exit'; PictureOff "ExitRuntime_KTP700_Basic_PN_TR"; PictureOn "ExitRuntime_KTP700_Basic_PN_TR"
      on Release: StopRuntime(0)
   Button "Template_Button" at 614,429 size 71x50; TextOff 'Text'
   Button "Template_Button_1" at 514,429 size 71x50; TextOff 'Text'
   Button "Template_Button_2" at 414,429 size 71x50; TextOff 'Text'
   Button "Template_Button_3" at 314,429 size 71x50; TextOff 'Text'
   Button "Template_Button_4" at 214,429 size 71x50; TextOff 'Text'
   Button "Template_Button_5" at 114,429 size 71x50; TextOff 'Text'
   Button "Start screen" at 14,429 size 71x50; TextOff 'Start screen'; PictureOff "NavigateHome_KTP700_Basic_PN_TR"; PictureOn "NavigateHome_KTP700_Basic_PN_TR"
      on Release: ActivateScreen("Restricted Access", 0)
   SymbolicIOField "Symbolic_IO_Field_Screen" at 93,9 size 600x33; TextOff '0'; TextOn '1'; TextList "TextList_ScreenNames"
      ProcessValue <- "Tag_ScreenNumber"
      on Change: ActivateScreenByNumber("Tag_ScreenNumber", 0)
   DateTimeField "HmiScreenItemData" at 695,25 size 105x25
   DateTimeField "HmiScreenItemData_1" at 695,0 size 105x25
   GraphicView "Logo" at 0,0 size 91x51; Picture "Logo of HMI_1"

screen "Operator Interface" 800x480
   on GenerateScreen: SetBit("PB_Automatic_HMI")
   on ClearScreen: ResetBit("PB_Automatic_HMI")
   Button "Button_1" at 286,116 size 200x96; TextOff 'Small Piece'
      on Press: SetBit("PB_Small_HMI")
      on Release: ResetBit("PB_Small_HMI")
   Button "Button_2" at 24,116 size 205x97; TextOff 'Large Piece'
      on Release: ResetBit("PB_Large_HMI")
      on Press: SetBit("PB_Large_HMI")
   Button "Button_4" at 285,230 size 202x90; TextOff 'Manual'
      on Press: SetBit("PB_Manual_HMI")
      on Release: ResetBit("PB_Manual_HMI")
   Button "Button_5" at 558,236 size 220x107; TextOff 'Stop Furnace'
      on Press: SetBit("PB_Furnace_Deactivation")
      on Release: ResetBit("PB_Furnace_Deactivation")
   Button "Button_3" at 559,18 size 219x200; TextOff 'Stop/Reset'
      on Press: SetBit("PB_Stop_HMI")
      on Release: ResetBit("PB_Stop_HMI")
   Button "Button_6" at 23,230 size 206x89; TextOff 'Automatic'
      on Press: SetBit("PB_Automatic_HMI")
   Button "Button_7" at 21,18 size 466x82; TextOff 'Funace Activation'
      on Press: SetBit("PB_Furnace_Activation")
      on Release: ResetBit("PB_Furnace_Activation")
   IOField "I/O field_1" at 24,360 size 106x37; FormatPattern s999999999.999
      ProcessValue <- "PID_Furnace_Control_Setpoint"
   TextField "Text field_1" at 21,332 size 227x23; Text 'Furnace Temp Setting (C°)'
   Button "Button_8" at 558,355 size 220x107; TextOff 'Monitoring'
      on Press: ActivateScreen("Process Monitoring", 0)
   Rectangle "Rectangle_1" at 286,343 size 203x120
      Appearance <- "System Enable"
   TextField "Text field_2" at 319,385 size 138x42; Text 'Automatic Mode Enabled'
   Button "Button_9" at 23,410 size 212x52; TextOff 'Restricted Access'
      on Press: ActivateScreen("Restricted Access", 0)

screen "Temperature History" 800x480
   TrendView "Trend view_1" at 29,18 size 484x444
   Button "Button_5" at 558,147 size 220x196; TextOff 'Stop Furnace'
      on Release: ResetBit("PB_Furnace_Deactivation")
      on Press: SetBit("PB_Furnace_Deactivation")
   Button "Button_8" at 558,355 size 220x107; TextOff 'Maintenance'
      on Press: ActivateScreen("Maintenance", 0)
   Button "Button_7" at 559,18 size 219x110; TextOff 'Funace Activation'
      on Release: ResetBit("PB_Furnace_Activation")
      on Press: SetBit("PB_Furnace_Activation")

screen "Management" 800x480
   IOField "I/O field_1" at 58,60 size 182x51; FormatPattern s99999
      ProcessValue <- "LargePart_Counter_0_DB_CV"
   IOField "I/O field_2" at 58,233 size 182x51; FormatPattern s99999
      ProcessValue <- "IEC_Total_Piece_Reject_Counter_0_DB_CV"
   IOField "I/O field_3" at 59,145 size 182x51; FormatPattern s99999
      ProcessValue <- "SmallPart_Counter_0_DB_CV"
   TextField "Text field_1" at 58,29 size 114x23; Text 'Large Pieces:'
   TextField "Text field_2" at 59,111 size 113x23; Text 'Small Pieces:'
   TextField "Text field_3" at 59,200 size 189x23; Text 'Total Pieces Rejected:'
   IOField "I/O field_4" at 58,319 size 182x51; FormatPattern s99999
      ProcessValue <- "IEC_Total_Error_Counter_0_DB_CV"
   TextField "Text field_4" at 58,287 size 108x23; Text 'Total Errors:'
   Button "Button_1" at 274,62 size 167x49; TextOff 'Reset'
      on Press: SetBit("PB_Reset_Counter_Large")
      on Release: ResetBit("PB_Reset_Counter_Large")
   Button "Button_2" at 274,147 size 167x49; TextOff 'Reset'
      on Release: ResetBit("PB_Reset_Counter_Small")
      on Press: SetBit("PB_Reset_Counter_Small")
   Button "Button_3" at 274,233 size 167x49; TextOff 'Reset'
      on Press: SetBit("PB_Reset_Counter_Rejects")
      on Release: ResetBit("PB_Reset_Counter_Rejects")
   Button "Button_4" at 274,319 size 167x49; TextOff 'Reset'
      on Release: ResetBit("PB_Reset_Counter_Errors")
      on Press: SetBit("PB_Reset_Counter_Errors")
   Button "Button_5" at 59,400 size 385x59; TextOff 'Reset All'
      on Press: SetBit("PB_Reset_Counter_All")
      on Release: ResetBit("PB_Reset_Counter_All")
   Button "Button_6" at 554,236 size 220x107; TextOff 'Stop Furnace'
      on Release: ResetBit("PB_Furnace_Deactivation")
      on Press: SetBit("PB_Furnace_Deactivation")
   Button "Button_7" at 555,18 size 219x200; TextOff 'Stop/Reset'
      on Release: ResetBit("PB_Stop_HMI")
      on Press: SetBit("PB_Stop_HMI")
   Button "Button_8" at 554,355 size 220x107; TextOff 'Back'
      on Press: function_efd93a16()

screen "Process Monitoring" 800x480
   Rectangle "Rectangle_1" at 27,40 size 137x59
      Appearance <- "Temp_in_Range"
   Rectangle "Rectangle_2" at 27,99 size 137x59
      Appearance <- "Piece_selected"
   Rectangle "Rectangle_3" at 27,158 size 137x59
      Appearance <- "System Enable"
   Rectangle "Rectangle_6" at 27,276 size 137x59
      Appearance <- "Furnace_Timer_0_DB_2_IN"
   TextField "Text field_1" at 43,58 size 96x23; Text 'Furnace On'
   TextField "Text field_2" at 42,107 size 88x42; Text 'Piece Size Selected'
   TextField "Text field_3" at 36,175 size 116x23; Text 'Automatic On'
   TextField "Text field_7" at 45,283 size 94x42; Text 'Furnace in Operation'
   Bar "Bar_1" at 193,40 size 77x412; MinimumValue 0; MaximumValue 450
      ProcessValue <- "PV_Memory"
   Button "Button_5" at 554,236 size 220x107; TextOff 'Stop Furnace'
      on Release: ResetBit("PB_Furnace_Deactivation")
      on Press: SetBit("PB_Furnace_Deactivation")
   Button "Button_3" at 555,18 size 219x200; TextOff 'Stop/Reset'
      on Release: ResetBit("PB_Stop_HMI")
      on Press: SetBit("PB_Stop_HMI")
   IOField "I/O field_1" at 283,227 size 106x37; FormatPattern s999999999.999
      ProcessValue <- "PID_Furnace_Control_Setpoint"
   TextField "Text field_8" at 281,192 size 163x23; Text 'Furnace Temp (C°)'
   IOField "I/O field_2" at 285,91 size 106x37; FormatPattern s999999999.999
      ProcessValue <- "Temp_High_Set_Point"
   TextField "Text field_9" at 285,57 size 238x23; Text 'Temp High Alarm Point (C°)'
   IOField "I/O field_3" at 281,377 size 106x37; FormatPattern s999999999.999
      ProcessValue <- "Temp_Low_Set_Point"
   TextField "Text field_10" at 278,343 size 234x23; Text 'Temp Low Alarm Point (C°)'
   Circle "Circle_1" at 416,377 size 39x39
      Appearance <- "Temp_Low_Alarm"
   Circle "Circle_2" at 418,86 size 39x39
      Appearance <- "Temp_High_Alarm"
   Circle "Circle_3" at 418,226 size 39x39
      Appearance <- "Temp_in_Range"
   Rectangle "Rectangle_4" at 27,217 size 137x59
      Appearance <- "Piece_Detected"
   TextField "Text field_4" at 36,232 size 119x23; Text 'Part Detected'
   Button "Button_8" at 554,355 size 220x107; TextOff 'Back'
      on Press: function_efd93a16()
   Button "Button_6" at 16,348 size 164x101; TextOff 'Automatic'
      on Press: SetBit("PB_Automatic_HMI")

screen "Restricted Access" 800x480
   Button "Button_1" at 97,55 size 269x236; TextOff 'Maintenance'
      on Press: ActivateScreen("Maintenance", 0)
   Button "Button_2" at 434,55 size 263x237; TextOff 'Management'
      on Click: ActivateScreen("Management", 0)
   Button "Button_8" at 97,314 size 600x107; TextOff 'Back to Controls'
      on Press: ActivateScreen("Operator Interface", 0)

screen "Maintenance" 800x480
   Button "Button_8" at 43,19 size 220x107; TextOff 'Monitoring'
      on Press: ActivateScreen("Process Monitoring", 0)
   Button "Button_1" at 298,18 size 220x107; TextOff 'Counters'
      on Press: ActivateScreen("Management", 0)
   Button "Button_5" at 554,236 size 220x107; TextOff 'Stop Furnace'
      on Release: ResetBit("PB_Furnace_Deactivation")
      on Press: SetBit("PB_Furnace_Deactivation")
   Button "Button_3" at 555,18 size 219x200; TextOff 'Stop/Reset'
      on Release: ResetBit("PB_Stop_HMI")
      on Press: SetBit("PB_Stop_HMI")
   Button "Button_2" at 554,355 size 220x107; TextOff 'Controls'
      on Press: ActivateScreen("Operator Interface", 0)
   IOField "I/O field_1" at 45,274 size 106x37; FormatPattern s999999999.999
      ProcessValue <- "PID_Furnace_Control_Setpoint"
   TextField "Text field_8" at 43,239 size 163x23; Text 'Furnace Temp (C°)'
   IOField "I/O field_2" at 43,192 size 106x37; FormatPattern s999999999.999
      ProcessValue <- "Temp_High_Set_Point"
   TextField "Text field_9" at 43,158 size 238x23; Text 'Temp High Alarm Point (C°)'
   Circle "Circle_2" at 181,186 size 39x39
      Appearance <- "Temp_High_Alarm"
   Circle "Circle_3" at 180,273 size 39x39
      Appearance <- "Temp_in_Range"
   IOField "I/O field_3" at 44,355 size 106x37; FormatPattern s999999999.999
      ProcessValue <- "Temp_Low_Set_Point"
   TextField "Text field_10" at 41,321 size 234x23; Text 'Temp Low Alarm Point (C°)'
   Circle "Circle_1" at 479,370 size 39x39
      Appearance <- "S3 Heat or Reject"
   Button "Button_4" at 298,149 size 220x107; TextOff 'Temperature History'
      on Press: ActivateScreen("Temperature History", 0)
   Circle "Circle_4" at 479,273 size 39x39
      Appearance <- "S1 Optical"
   Circle "Circle_6" at 479,321 size 39x39
      Appearance <- "S2 Optical"
   TextField "Text field_1" at 437,323 size 35x32; Text 'S2'
   TextField "Text field_2" at 437,273 size 35x32; Text 'S1'
   TextField "Text field_3" at 437,374 size 35x32; Text 'S3'
   Circle "Circle_8" at 479,423 size 39x39
      Appearance <- "Piece_inserted_Error_Light_HMI"
   TextField "Text field_4" at 215,423 size 257x32; Text 'Error Piece in Process'
   Circle "Circle_9" at 180,355 size 39x39
      Appearance <- "Temp_Low_Alarm"
*)